PROGRAM P_Demo_FB_DMXGetDMX512PersonalityDescription
VAR
    fbGetPersDesc     : FB_DMXGetDMX512PersonalityDescription; // 读 personality 描述
    stDmxCmdBuffer    : ST_DMXCommandBuffer;          // 与通讯 FB 共用
    wTargetManufId    : WORD := 16#4241;              // 目标灯具厂商 ID
    dwTargetDeviceId  : DWORD := 16#12131415;         // 目标灯具设备 ID
    byTargetPort      : BYTE := 0;                    // 根设备通道 0
    byWantPersonality : BYTE := 1;                    // 查询 personality 1
    bDoRead           : BOOL := FALSE;                // 在线给一次上升沿触发
    bBusy             : BOOL;
    bError            : BOOL;
    udiErrId          : UDINT;
    stPersDesc        : ST_DMX512PersonalityDescription;  // personality 描述
END_VAR

// ============================================================
// Tc2_DMX.FB_DMXGetDMX512PersonalityDescription 演示程序
// ============================================================
// 场景：为多模式灯具选工作模式：遍历各 personality 描述(看占多少通道/功能)，据现场通道预算选定。
// 价值：把各工作模式占用通道数与说明读出集中比较，避免凭手册猜测、选错模式导致通道冲突。
// 验证：设 byWantPersonality:=1，给 bDoRead 一次上升沿 -> bBusy 短暂 TRUE -> 回 FALSE 后 stPersDesc 含该 personality 占用槽数与文本说明。
// 验证步骤：
//   1. 右键 PLC 项目下 POUs 文件夹 → Add → Existing Item → 选本 .TcPOU 文件
//   2. 引用 Tc2_DMX；同项目里放一个 FB_EL6851CommunicationEx 实例并共用 stDmxCmdBuffer（非 CycleMode）
//   3. 编译 → 登录 → 运行；按上方『验证』行在线给上升沿观察
// ============================================================

fbGetPersDesc(
    bStart                     := bDoRead,
    wDestinationManufacturerId := wTargetManufId,
    dwDestinationDeviceId      := dwTargetDeviceId,
    byPortId                   := byTargetPort,
    byPersonality              := byWantPersonality,
    dwOptions                  := 0,
    stCommandBuffer            := stDmxCmdBuffer,
    bBusy                      => bBusy,
    bError                     => bError,
    udiErrorId                 => udiErrId,
    stDMX512PersonalityDescription => stPersDesc
);

END_PROGRAM

(* stored: Version 1.1.0.1, ProductVersion 3.1.4024.5
   POU P_Demo_FB_DMXGetDMX512PersonalityDescription: Id {25534bf8-658c-5cc8-a60a-3be0fc30582a}, SpecialFunc None *)
